FUNCTION_BLOCK overcurrent_1 (* Composite Function Block Type *)
  (* Standard: 61499-2 *)
  (* Version 0.0, 22/03/2016, Chen-Wei, nxtControl GmbH, template *)
  PACKAGE Main;
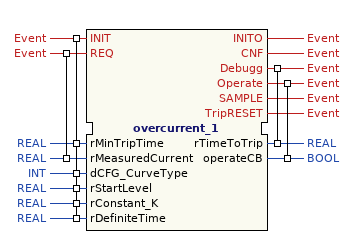
  EVENT_INPUT
    INIT WITH rMinTripTime, dCFG_CurveType, rStartLevel, rConstant_K, rDefiniteTime; (* Initialization Request *)
    REQ WITH rMeasuredCurrent; (* Normal Execution Request *)
  END_EVENT
  EVENT_OUTPUT
    INITO; (* Initialization Confirm *)
    CNF; (* Execution Confirmation *)
    Debugg WITH rTimeToTrip;
    Operate WITH operateCB; (* Delayed Event *)
    SAMPLE;
    TripRESET;
  END_EVENT
  VAR_INPUT
    rMinTripTime : REAL; (* Input event qualifier *)
    rMeasuredCurrent : REAL; (* Input event qualifier *)
    dCFG_CurveType : INT;
    rStartLevel : REAL;
    rConstant_K : REAL;
    rDefiniteTime : REAL;
  END_VAR
  VAR_OUTPUT
    rTimeToTrip : REAL;
    operateCB : BOOL; (* Output event qualifier *)
  END_VAR
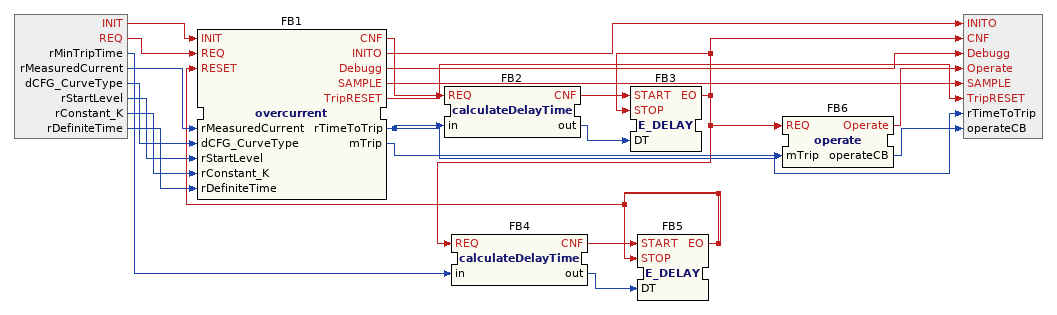
  FBS
    FB2 : calculateDelayTime;
    FB3 : E_DELAY;
    FB4 : calculateDelayTime;
    FB5 : E_DELAY;
    FB6 : operate;
    FB1 : overcurrent;
  END_FBS
  EVENT_CONNECTIONS
    FB1.CNF TO FB2.REQ;
    FB2.CNF TO FB3.START;
    FB3.EO TO FB3.STOP;
    FB4.CNF TO FB5.START;
    FB5.EO TO FB5.STOP;
    FB3.EO TO FB4.REQ;
    INIT TO FB1.INIT;
    REQ TO FB1.REQ;
    FB1.INITO TO INITO;
    FB1.Debugg TO Debugg;
    FB3.EO TO FB6.REQ;
    FB6.Operate TO Operate;
    FB5.EO TO FB1.RESET;
    FB1.SAMPLE TO SAMPLE;
    FB1.TripRESET TO TripRESET;
    FB3.EO TO CNF;
  END_CONNECTIONS
  DATA_CONNECTIONS
    FB1.rTimeToTrip TO FB2.in;
    FB2.out TO FB3.DT;
    FB4.out TO FB5.DT;
    rMinTripTime TO FB4.in;
    rMeasuredCurrent TO FB1.rMeasuredCurrent;
    dCFG_CurveType TO FB1.dCFG_CurveType;
    rStartLevel TO FB1.rStartLevel;
    rConstant_K TO FB1.rConstant_K;
    rDefiniteTime TO FB1.rDefiniteTime;
    FB1.rTimeToTrip TO rTimeToTrip;
    FB1.mTrip TO FB6.mTrip;
    FB6.operateCB TO operateCB;
  END_CONNECTIONS
END_FUNCTION_BLOCK
